(* IEC 61131-3 sources: RL_MAR/experiments/comparison/llm4plc/results/gpt-4o-mini_20260506_100619/20260506_100719, 3 files *)

(* ---- generated_code_iteration_0.st ---- *)
ructured-text
FUNCTION_BLOCK SelectSort
VAR_INPUT
    exe : BOOL;
    seq : VARIANT;
END_VAR
VAR_OUTPUT
    error : BOOL;
    status : WORD;
END_VAR
VAR
    arrayLength : INT; // Length of the array
    i : INT; // Loop variable for outer loop
    j : INT; // Loop variable for inner loop
    temp : VARIANT; // Temporary variable for swapping
    isArray : BOOL; // Flag to check if seq is an array type
END_VAR

// State initialization
IF exe THEN
    error := FALSE;
    status := 16#0000; // No error
    isArray := FALSE;

    // Check if seq is an array type
    IF (TypeOf(seq) = ARRAY) THEN
        isArray := TRUE;
        arrayLength := ARRAY_LENGTH(seq); // Get the length of the array
    ELSE
        error := TRUE;
        status := 16#8A01; // Invalid array type
    END_IF;

    // Perform sorting if seq is a valid array type
    IF isArray THEN
        // Selection sort algorithm
        FOR i := 0 TO arrayLength - 2 DO
            // Assume the minimum is the first element
            VAR minIndex : INT := i;
            FOR j := i + 1 TO arrayLength - 1 DO
                // Find the minimum element in the unsorted array
                IF seq[j] < seq[minIndex] THEN
                    minIndex := j;
                END_IF;
            END_FOR;

            // Swap the found minimum element with the first element
            IF minIndex <> i THEN
                temp := seq[i];
                seq[i] := seq[minIndex];
                seq[minIndex] := temp;
            END_IF;
        END_FOR;
    END_IF;

    // Finalize sorting process
    IF NOT error THEN
        error := FALSE;
        status := 16#0000; // No error
    END_IF;
END_IF;

END_FUNCTION_BLOCK

(* ---- generated_code_iteration_1.st ---- *)
START_REASON
The errors in the original Structured Text (ST) code were primarily due to the use of the 'VARIANT' type, which is not recognized in the context of the CODESYS compiler. This type is often not supported in many PLC programming environments, leading to compilation errors. Additionally, the code structure needs to adhere to the proper syntax and conventions of Structured Text, particularly in variable declaration and handling.

To correct these errors, I will replace the 'VARIANT' type with a more specific type that is compatible with CODESYS, such as an array of integers (or another appropriate type based on the intended use). I will also ensure that the variable sections are properly closed with "END_VAR" and maintain the function block structure as required.
END_REASON

START_ST
FUNCTION_BLOCK SelectSort
VAR_INPUT
    exe : BOOL;
    seq : ARRAY[0..99] OF INT; // Assuming the array is of type INT with a maximum length of 100
END_VAR
VAR_OUTPUT
    error : BOOL;
    status : WORD;
END_VAR
VAR
    arrayLength : INT; // Length of the array
    i : INT; // Loop variable for outer loop
    j : INT; // Loop variable for inner loop
    temp : INT; // Temporary variable for swapping
    isArray : BOOL; // Flag to check if seq is an array type
END_VAR

// State initialization
IF exe THEN
    error := FALSE;
    status := 16#0000; // No error
    isArray := TRUE; // Since we are using a defined array type

    // Get the length of the array
    arrayLength := SIZEOF(seq) / SIZEOF(seq[0]); // Calculate the number of elements in the array

    // Perform sorting if seq is a valid array type
    IF isArray THEN
        // Selection sort algorithm
        FOR i := 0 TO arrayLength - 2 DO
            // Assume the minimum is the first element
            VAR minIndex : INT := i;
            FOR j := i + 1 TO arrayLength - 1 DO
                // Find the minimum element in the unsorted array
                IF seq[j] < seq[minIndex] THEN
                    minIndex := j;
                END_IF;
            END_FOR;

            // Swap the found minimum element with the first element
            IF minIndex <> i THEN
                temp := seq[i];
                seq[i] := seq[minIndex];
                seq[minIndex] := temp;
            END_IF;
        END_FOR;
    END_IF;

    // Finalize sorting process
    IF NOT error THEN
        error := FALSE;
        status := 16#0000; // No error
    END_IF;
END_IF;

END_FUNCTION_BLOCK
END_ST

(* ---- generated_code_iteration_2.st ---- *)
START_REASON
The errors in the original Structured Text (ST) code were primarily due to the incorrect placement of the variable declaration section. The CODESYS compiler does not allow variable declarations to be nested within the main execution block of the function block. All variable declarations must be placed in the appropriate sections defined at the beginning of the function block.

To correct these errors, I will ensure that all variable declarations are properly placed in the VAR section and that the code adheres to the correct syntax. I will also ensure that the sorting logic remains intact and that the overall structure of the function block is maintained without any nesting of variable declarations within the execution logic.

END_REASON

START_ST
FUNCTION_BLOCK SelectSort
VAR_INPUT
    exe : BOOL;
    seq : ARRAY[0..99] OF INT; // Assuming the array is of type INT with a maximum length of 100
END_VAR
VAR_OUTPUT
    error : BOOL;
    status : WORD;
END_VAR
VAR
    arrayLength : INT; // Length of the array
    i : INT; // Loop variable for outer loop
    j : INT; // Loop variable for inner loop
    temp : INT; // Temporary variable for swapping
    minIndex : INT; // Variable to hold the index of the minimum element
END_VAR

// State initialization
IF exe THEN
    error := FALSE;
    status := 16#0000; // No error

    // Get the length of the array
    arrayLength := SIZEOF(seq) / SIZEOF(seq[0]); // Calculate the number of elements in the array

    // Selection sort algorithm
    FOR i := 0 TO arrayLength - 2 DO
        // Assume the minimum is the first element
        minIndex := i;
        FOR j := i + 1 TO arrayLength - 1 DO
            // Find the minimum element in the unsorted array
            IF seq[j] < seq[minIndex] THEN
                minIndex := j;
            END_IF;
        END_FOR;

        // Swap the found minimum element with the first element
        IF minIndex <> i THEN
            temp := seq[i];
            seq[i] := seq[minIndex];
            seq[minIndex] := temp;
        END_IF;
    END_FOR;

    // Finalize sorting process
    IF NOT error THEN
        error := FALSE;
        status := 16#0000; // No error
    END_IF;
END_IF;

END_FUNCTION_BLOCK
END_ST
